Staubli VAL3: start.pgx

program start()
  local num l_nIndex
begin
  resetMotion()
  movej(jStart, tTool, mRapide100)

  // paramètrage du server tcp
  sioCtrl(sData, "port", 8500)
  sioCtrl(sData, "clients", 1)
  //CCaractère de fin de line : Line Feed
  sioCtrl(sData, "endOfString", 13)



  logMsg("------------ Sio Initialise")

  //  Créé des taches pour le multi-threading, Prio 50 = neutre
  while true

    if !bAcquisitionOk
      call dataAcquisition()
    else
      call goToPoint()
    endIf

  endWhile

  waitEndMove()
end
